LIN {X 0,Y 97.442,Z 457.914,A -85,B 0,C 180,E1 -28297.811,E2 -28297.811} C_VEL
LIN {X 0,Y 89.489,Z 462.022,A -85,B 0,C 180,E1 -28300.482,E2 -28300.482} C_VEL
LIN {X 0,Y 81.671,Z 465.606,A -85,B 0,C 180,E1 -28303.794,E2 -28303.794} C_VEL
LIN {X 0,Y 77.924,Z 467.495,A -85,B 0,C 180,E1 -28306.759,E2 -28306.759} C_VEL
LIN {X 0,Y 72.015,Z 470.678,A -85,B 0,C 180,E1 -28314.162,E2 -28314.162} C_VEL
LIN {X 0,Y 66.399,Z 473.568,A -85,B 0,C 180,E1 -28324.955,E2 -28324.955} C_VEL
LIN {X 0,Y 63.238,Z 475.299,A -85,B 0,C 180,E1 -28337.16,E2 -28337.16} C_VEL
LIN {X 0,Y 62.547,Z 475.896,A -85,B 0,C 180,E1 -28350.002,E2 -28350.002} C_VEL
LIN {X 0,Y 63.235,Z 475.326,A -85,B 0,C 180,E1 -28362.845,E2 -28362.845} C_VEL
LIN {X 0,Y 66.353,Z 473.633,A -85,B 0,C 180,E1 -28375.069,E2 -28375.069} C_VEL
LIN {X 0,Y 71.978,Z 470.774,A -85,B 0,C 180,E1 -28385.865,E2 -28385.865} C_VEL
LIN {X 0,Y 79.628,Z 466.628,A -85,B 0,C 180,E1 -28395.082,E2 -28395.082} C_VEL
LIN {X 0,Y 88.746,Z 461.261,A -85,B 0,C 180,E1 -28402.367,E2 -28402.367} C_VEL
LIN {X 0,Y 99.079,Z 454.353,A -85,B 0,C 180,E1 -28408.344,E2 -28408.344} C_VEL
LIN {X 0,Y 108.881,Z 446.931,A -85,B 0,C 180,E1 -28412.566,E2 -28412.566} C_VEL
LIN {X 0,Y 119.077,Z 437.984,A -85,B 0,C 180,E1 -28416.181,E2 -28416.181} C_VEL
LIN {X 0,Y 123.43,Z 433.764,A -85,B 0,C 180,E1 -28417.473,E2 -28417.473} C_VEL
LIN {X 0,Y 124.559,Z 432.45,A -85,B 0,C 180,E1 -28418.106,E2 -28418.106} C_VEL
LIN {X 0,Y 125.877,Z 428.922,A -85,B 0,C 180,E1 -28421.651,E2 -28421.651} C_VEL
LIN {X 0,Y 126.554,Z 427.011,A -85,B 0,C 180,E1 -28423.879,E2 -28423.879} C_VEL
LIN {X 0,Y 126.966,Z 424.818,A -85,B 0,C 180,E1 -28427.208,E2 -28427.208} C_VEL
LIN {X 0,Y 127.18,Z 423.255,A -85,B 0,C 180,E1 -28430.457,E2 -28430.457} C_VEL
LIN {X 0,Y 127.338,Z 422.165,A -85,B 0,C 180,E1 -28433.662,E2 -28433.662} C_VEL
LIN {X 0,Y 127.868,Z 420.898,A -85,B 0,C 180,E1 -28440,E2 -28440} C_VEL
LIN {X 0,Y 127.415,Z 422.493,A -85,B 0,C 180,E1 -28446.852,E2 -28446.852} C_VEL
LIN {X 0,Y 127.255,Z 423.571,A -85,B 0,C 180,E1 -28449.537,E2 -28449.537} C_VEL
LIN {X 0,Y 126.822,Z 425.492,A -85,B 0,C 180,E1 -28452.806,E2 -28452.806} C_VEL
LIN {X 0,Y 126.028,Z 428.183,A -85,B 0,C 180,E1 -28456.19,E2 -28456.19} C_VEL
LIN {X 0,Y 124.785,Z 431.569,A -85,B 0,C 180,E1 -28459.75,E2 -28459.75} C_VEL
LIN {X 0,Y 123.924,Z 433.592,A -85,B 0,C 180,E1 -28461.568,E2 -28461.568} C_VEL
LIN {X 0,Y 122.983,Z 434.784,A -85,B 0,C 180,E1 -28462.222,E2 -28462.222} C_VEL
LIN {X 0,Y 112.81,Z 444.196,A -85,B 0,C 180,E1 -28465.398,E2 -28465.398} C_VEL
LIN {X 0,Y 104.198,Z 451.23,A -85,B 0,C 180,E1 -28468.736,E2 -28468.736} C_VEL
LIN {X 0,Y 96.042,Z 457.197,A -85,B 0,C 180,E1 -28472.697,E2 -28472.697} C_VEL
LIN {X 0,Y 85.88,Z 463.77,A -85,B 0,C 180,E1 -28478.972,E2 -28478.972} C_VEL
LIN {X 0,Y 76.763,Z 469.049,A -85,B 0,C 180,E1 -28487.09,E2 -28487.09} C_VEL
LIN {X 0,Y 71.544,Z 471.892,A -85,B 0,C 180,E1 -28493.884,E2 -28493.884} C_VEL
LIN {X 0,Y 66.002,Z 474.79,A -85,B 0,C 180,E1 -28504.789,E2 -28504.789} C_VEL
LIN {X 0,Y 63.046,Z 476.52,A -85,B 0,C 180,E1 -28517.115,E2 -28517.115} C_VEL
LIN {X 0,Y 62.488,Z 477.112,A -85,B 0,C 180,E1 -28529.998,E2 -28529.998} C_VEL
LIN {X 0,Y 63.044,Z 476.499,A -85,B 0,C 180,E1 -28542.88,E2 -28542.88} C_VEL
LIN {X 0,Y 66.001,Z 474.741,A -85,B 0,C 180,E1 -28555.207,E2 -28555.207} C_VEL
LIN {X 0,Y 71.552,Z 471.819,A -85,B 0,C 180,E1 -28566.106,E2 -28566.106} C_VEL
LIN {X 0,Y 79.126,Z 467.663,A -85,B 0,C 180,E1 -28575.277,E2 -28575.277} C_VEL
LIN {X 0,Y 88.295,Z 462.161,A -85,B 0,C 180,E1 -28582.743,E2 -28582.743} C_VEL
LIN {X 0,Y 98.752,Z 455.167,A -85,B 0,C 180,E1 -28588.647,E2 -28588.647} C_VEL
LIN {X 0,Y 108.712,Z 447.473,A -85,B 0,C 180,E1 -28593.094,E2 -28593.094} C_VEL
LIN {X 0,Y 118.744,Z 438.664,A -85,B 0,C 180,E1 -28596.541,E2 -28596.541} C_VEL
LIN {X 0,Y 122.944,Z 434.565,A -85,B 0,C 180,E1 -28597.783,E2 -28597.783} C_VEL
LIN {X 0,Y 123.888,Z 433.395,A -85,B 0,C 180,E1 -28598.402,E2 -28598.402} C_VEL
LIN {X 0,Y 125.435,Z 429.38,A -85,B 0,C 180,E1 -28602.262,E2 -28602.262} C_VEL
LIN {X 0,Y 126.427,Z 426.495,A -85,B 0,C 180,E1 -28605.514,E2 -28605.514} C_VEL
LIN {X 0,Y 126.719,Z 425.289,A -85,B 0,C 180,E1 -28607.183,E2 -28607.183} C_VEL
LIN {X 0,Y 127.153,Z 423.361,A -85,B 0,C 180,E1 -28610.456,E2 -28610.456} C_VEL
LIN {X 0,Y 127.373,Z 422.07,A -85,B 0,C 180,E1 -28613.665,E2 -28613.665} C_VEL
LIN {X 0,Y 127.794,Z 420.619,A -85,B 0,C 180,E1 -28620,E2 -28620} C_VEL
LIN {X 0,Y 127.238,Z 421.924,A -85,B 0,C 180,E1 -28626.343,E2 -28626.343} C_VEL
LIN {X 0,Y 127.08,Z 423.01,A -85,B 0,C 180,E1 -28629.551,E2 -28629.551} C_VEL
LIN {X 0,Y 126.764,Z 425.502,A -85,B 0,C 180,E1 -28634.448,E2 -28634.448} C_VEL
LIN {X 0,Y 125.828,Z 428.596,A -85,B 0,C 180,E1 -28638.29,E2 -28638.29} C_VEL
LIN {X 0,Y 124.488,Z 432.184,A -85,B 0,C 180,E1 -28641.887,E2 -28641.887} C_VEL
LIN {X 0,Y 123.467,Z 433.483,A -85,B 0,C 180,E1 -28642.608,E2 -28642.608} C_VEL
LIN {X 0,Y 114.3,Z 442.123,A -85,B 0,C 180,E1 -28645.494,E2 -28645.494} C_VEL
LIN {X 0,Y 103.312,Z 451.121,A -85,B 0,C 180,E1 -28649.853,E2 -28649.853} C_VEL
LIN {X 0,Y 93.855,Z 457.813,A -85,B 0,C 180,E1 -28654.548,E2 -28654.548} C_VEL
LIN {X 0,Y 84.04,Z 464.002,A -85,B 0,C 180,E1 -28661.184,E2 -28661.184} C_VEL
LIN {X 0,Y 77.924,Z 467.495,A -85,B 0,C 180,E1 -28666.759,E2 -28666.759} C_VEL
LIN {X 0,Y 74.365,Z 469.237,A -85,B 0,C 180,E1 -28670.048,E2 -28670.048} C_VEL
LIN {X 0,Y 67.326,Z 471.662,A -85,B 0,C 180,E1 -28675.354,E2 -28675.354} C_VEL
LIN {X 0,Y 60.799,Z 473.558,A -85,B 0,C 180,E1 -28681.878,E2 -28681.878} C_VEL
LIN {X 0,Y 58.285,Z 474.398,A -85,B 0,C 180,E1 -28686.971,E2 -28686.971} C_VEL
LIN {X 0,Y 56.319,Z 475.368,A -85,B 0,C 180,E1 -28695.55,E2 -28695.55} C_VEL
LIN {X 0,Y 55.465,Z 475.965,A -85,B 0,C 180,E1 -28710.003,E2 -28710.003} C_VEL
LIN {X 0,Y 56.315,Z 475.395,A -85,B 0,C 180,E1 -28724.456,E2 -28724.456} C_VEL
LIN {X 0,Y 59.949,Z 473.702,A -85,B 0,C 180,E1 -28737.967,E2 -28737.967} C_VEL
LIN {X 0,Y 66.327,Z 470.843,A -85,B 0,C 180,E1 -28749.479,E2 -28749.479} C_VEL
LIN {X 0,Y 74.653,Z 466.753,A -85,B 0,C 180,E1 -28758.865,E2 -28758.865} C_VEL
LIN {X 0,Y 84.571,Z 461.329,A -85,B 0,C 180,E1 -28766.205,E2 -28766.205} C_VEL
LIN {X 0,Y 95.532,Z 454.42,A -85,B 0,C 180,E1 -28771.984,E2 -28771.984} C_VEL
LIN {X 0,Y 105.763,Z 446.999,A -85,B 0,C 180,E1 -28776.022,E2 -28776.022} C_VEL
LIN {X 0,Y 116.379,Z 438.051,A -85,B 0,C 180,E1 -28779.396,E2 -28779.396} C_VEL
LIN {X 0,Y 119.463,Z 435.151,A -85,B 0,C 180,E1 -28780.269,E2 -28780.269} C_VEL
LIN {X 0,Y 120.636,Z 432.702,A -85,B 0,C 180,E1 -28783.064,E2 -28783.064} C_VEL
LIN {X 0,Y 121.277,Z 431.216,A -85,B 0,C 180,E1 -28784.884,E2 -28784.884} C_VEL
LIN {X 0,Y 121.641,Z 430.076,A -85,B 0,C 180,E1 -28786.637,E2 -28786.637} C_VEL
LIN {X 0,Y 121.963,Z 428.494,A -85,B 0,C 180,E1 -28790.045,E2 -28790.045} C_VEL
LIN {X 0,Y 122.275,Z 427.316,A -85,B 0,C 180,E1 -28793.399,E2 -28793.399} C_VEL
LIN {X 0,Y 122.896,Z 426.011,A -85,B 0,C 180,E1 -28800,E2 -28800} C_VEL
LIN {X 0,Y 122.378,Z 427.479,A -85,B 0,C 180,E1 -28806.595,E2 -28806.595} C_VEL
LIN {X 0,Y 121.745,Z 429.512,A -85,B 0,C 180,E1 -28811.077,E2 -28811.077} C_VEL
LIN {X 0,Y 121.308,Z 430.918,A -85,B 0,C 180,E1 -28813.399,E2 -28813.399} C_VEL
LIN {X 0,Y 119.986,Z 433.936,A -85,B 0,C 180,E1 -28817.029,E2 -28817.029} C_VEL
LIN {X 0,Y 119.037,Z 435.896,A -85,B 0,C 180,E1 -28819.152,E2 -28819.152} C_VEL
LIN {X 0,Y 117.658,Z 437.389,A -85,B 0,C 180,E1 -28819.815,E2 -28819.815} C_VEL
LIN {X 0,Y 106.892,Z 446.596,A -85,B 0,C 180,E1 -28823.003,E2 -28823.003} C_VEL
LIN {X 0,Y 96.663,Z 454.257,A -85,B 0,C 180,E1 -28827.043,E2 -28827.043} C_VEL
LIN {X 0,Y 86.828,Z 460.604,A -85,B 0,C 180,E1 -28831.799,E2 -28831.799} C_VEL
LIN {X 0,Y 76.579,Z 466.441,A -85,B 0,C 180,E1 -28838.73,E2 -28838.73} C_VEL
LIN {X 0,Y 69.824,Z 469.915,A -85,B 0,C 180,E1 -28845.203,E2 -28845.203} C_VEL
LIN {X 0,Y 62.467,Z 473.422,A -85,B 0,C 180,E1 -28855.766,E2 -28855.766} C_VEL
LIN {X 0,Y 57.49,Z 475.729,A -85,B 0,C 180,E1 -28868.483,E2 -28868.483} C_VEL
LIN {X 0,Y 55.392,Z 476.889,A -85,B 0,C 180,E1 -28882.708,E2 -28882.708} C_VEL
LIN {X 0,Y 55.387,Z 477.043,A -85,B 0,C 180,E1 -28889.997,E2 -28889.997} C_VEL
LIN {X 0,Y 56.105,Z 476.429,A -85,B 0,C 180,E1 -28904.506,E2 -28904.506} C_VEL
LIN {X 0,Y 59.603,Z 474.671,A -85,B 0,C 180,E1 -28918.138,E2 -28918.138} C_VEL
LIN {X 0,Y 65.896,Z 471.749,A -85,B 0,C 180,E1 -28929.781,E2 -28929.781} C_VEL
LIN {X 0,Y 74.266,Z 467.592,A -85,B 0,C 180,E1 -28939.202,E2 -28939.202} C_VEL
LIN {X 0,Y 84.154,Z 462.09,A -85,B 0,C 180,E1 -28946.625,E2 -28946.625} C_VEL
LIN {X 0,Y 95.235,Z 455.096,A -85,B 0,C 180,E1 -28952.315,E2 -28952.315} C_VEL
LIN {X 0,Y 104.959,Z 447.945,A -85,B 0,C 180,E1 -28956.312,E2 -28956.312} C_VEL
LIN {X 0,Y 116.087,Z 438.592,A -85,B 0,C 180,E1 -28959.776,E2 -28959.776} C_VEL
LIN {X 0,Y 117.64,Z 437.143,A -85,B 0,C 180,E1 -28960.201,E2 -28960.201} C_VEL
LIN {X 0,Y 118.973,Z 435.649,A -85,B 0,C 180,E1 -28960.93,E2 -28960.93} C_VEL
LIN {X 0,Y 120.601,Z 432.176,A -85,B 0,C 180,E1 -28964.798,E2 -28964.798} C_VEL
LIN {X 0,Y 121.203,Z 430.735,A -85,B 0,C 180,E1 -28966.589,E2 -28966.589} C_VEL
LIN {X 0,Y 121.854,Z 428.703,A -85,B 0,C 180,E1 -28970.036,E2 -28970.036} C_VEL
LIN {X 0,Y 122.294,Z 427.252,A -85,B 0,C 180,E1 -28973.4,E2 -28973.4} C_VEL
LIN {X 0,Y 122.823,Z 425.753,A -85,B 0,C 180,E1 -28980,E2 -28980} C_VEL
LIN {X 0,Y 122.169,Z 427.091,A -85,B 0,C 180,E1 -28986.607,E2 -28986.607} C_VEL
LIN {X 0,Y 121.743,Z 428.758,A -85,B 0,C 180,E1 -28991.085,E2 -28991.085} C_VEL
LIN {X 0,Y 121.552,Z 429.836,A -85,B 0,C 180,E1 -28993.373,E2 -28993.373} C_VEL
LIN {X 0,Y 120.585,Z 432.443,A -85,B 0,C 180,E1 -28996.943,E2 -28996.943} C_VEL
LIN {X 0,Y 119.411,Z 434.854,A -85,B 0,C 180,E1 -28999.67,E2 -28999.67} C_VEL
LIN {X 0,Y 116.428,Z 437.778,A -85,B 0,C 180,E1 -29000.675,E2 -29000.675} C_VEL
LIN {X 0,Y 105.837,Z 446.761,A -85,B 0,C 180,E1 -29004.075,E2 -29004.075} C_VEL
LIN {X 0,Y 95.571,Z 454.208,A -85,B 0,C 180,E1 -29008.066,E2 -29008.066} C_VEL
LIN {X 0,Y 84.625,Z 461.165,A -85,B 0,C 180,E1 -29013.856,E2 -29013.856} C_VEL
LIN {X 0,Y 74.274,Z 466.832,A -85,B 0,C 180,E1 -29021.481,E2 -29021.481} C_VEL
LIN {X 0,Y 66.361,Z 470.748,A -85,B 0,C 180,E1 -29030.552,E2 -29030.552} C_VEL
LIN {X 0,Y 59.992,Z 473.638,A -85,B 0,C 180,E1 -29042.06,E2 -29042.06} C_VEL
LIN {X 0,Y 58.285,Z 474.398,A -85,B 0,C 180,E1 -29046.971,E2 -29046.971} C_VEL
LIN {X 0,Y 56.244,Z 475.136,A -85,B 0,C 180,E1 -29052.47,E2 -29052.47} C_VEL
LIN {X 0,Y 53.738,Z 475.668,A -85,B 0,C 180,E1 -29058.065,E2 -29058.065} C_VEL
LIN {X 0,Y 49.32,Z 476.068,A -85,B 0,C 180,E1 -29070.536,E2 -29070.536} C_VEL
LIN {X 0,Y 48.601,Z 475.81,A -85,B 0,C 180,E1 -29079.882,E2 -29079.882} C_VEL
LIN {X 0,Y 51.219,Z 474.76,A -85,B 0,C 180,E1 -29094.311,E2 -29094.311} C_VEL
LIN {X 0,Y 57.045,Z 472.491,A -85,B 0,C 180,E1 -29108.027,E2 -29108.027} C_VEL
LIN {X 0,Y 65.36,Z 469.026,A -85,B 0,C 180,E1 -29118.827,E2 -29118.827} C_VEL
LIN {X 0,Y 75.354,Z 464.284,A -85,B 0,C 180,E1 -29127.079,E2 -29127.079} C_VEL
LIN {X 0,Y 86.504,Z 458.141,A -85,B 0,C 180,E1 -29133.343,E2 -29133.343} C_VEL
LIN {X 0,Y 98.494,Z 450.406,A -85,B 0,C 180,E1 -29138.068,E2 -29138.068} C_VEL
LIN {X 0,Y 109.411,Z 442.08,A -85,B 0,C 180,E1 -29141.538,E2 -29141.538} C_VEL
LIN {X 0,Y 114.064,Z 438.118,A -85,B 0,C 180,E1 -29142.752,E2 -29142.752} C_VEL
LIN {X 0,Y 115.111,Z 436.741,A -85,B 0,C 180,E1 -29144.021,E2 -29144.021} C_VEL
LIN {X 0,Y 115.899,Z 435.266,A -85,B 0,C 180,E1 -29145.985,E2 -29145.985} C_VEL
LIN {X 0,Y 116.535,Z 433.504,A -85,B 0,C 180,E1 -29149.576,E2 -29149.576} C_VEL
LIN {X 0,Y 116.94,Z 432.294,A -85,B 0,C 180,E1 -29153.096,E2 -29153.096} C_VEL
LIN {X 0,Y 117.708,Z 430.931,A -85,B 0,C 180,E1 -29160,E2 -29160} C_VEL
LIN {X 0,Y 117.302,Z 431.567,A -85,B 0,C 180,E1 -29163.434,E2 -29163.434} C_VEL
LIN {X 0,Y 117.008,Z 432.494,A -85,B 0,C 180,E1 -29166.899,E2 -29166.899} C_VEL
LIN {X 0,Y 116.402,Z 434.014,A -85,B 0,C 180,E1 -29170.435,E2 -29170.435} C_VEL
LIN {X 0,Y 115.253,Z 436.366,A -85,B 0,C 180,E1 -29174.117,E2 -29174.117} C_VEL
LIN {X 0,Y 113.826,Z 438.748,A -85,B 0,C 180,E1 -29176.857,E2 -29176.857} C_VEL
LIN {X 0,Y 102.087,Z 448.202,A -85,B 0,C 180,E1 -29180.041,E2 -29180.041} C_VEL
LIN {X 0,Y 92.127,Z 455.199,A -85,B 0,C 180,E1 -29183.731,E2 -29183.731} C_VEL
LIN {X 0,Y 80.455,Z 462.152,A -85,B 0,C 180,E1 -29189.127,E2 -29189.127} C_VEL
LIN {X 0,Y 69.762,Z 467.619,A -85,B 0,C 180,E1 -29196.296,E2 -29196.296} C_VEL
LIN {X 0,Y 60.555,Z 471.754,A -85,B 0,C 180,E1 -29205.861,E2 -29205.861} C_VEL
LIN {X 0,Y 53.399,Z 474.652,A -85,B 0,C 180,E1 -29218.231,E2 -29218.231} C_VEL
LIN {X 0,Y 49.236,Z 476.382,A -85,B 0,C 180,E1 -29233.409,E2 -29233.409} C_VEL
LIN {X 0,Y 48.302,Z 476.974,A -85,B 0,C 180,E1 -29249.997,E2 -29249.997} C_VEL
LIN {X 0,Y 49.234,Z 476.36,A -85,B 0,C 180,E1 -29266.585,E2 -29266.585} C_VEL
LIN {X 0,Y 53.398,Z 474.601,A -85,B 0,C 180,E1 -29281.762,E2 -29281.762} C_VEL
LIN {X 0,Y 60.563,Z 471.678,A -85,B 0,C 180,E1 -29294.123,E2 -29294.123} C_VEL
LIN {X 0,Y 69.785,Z 467.521,A -85,B 0,C 180,E1 -29303.671,E2 -29303.671} C_VEL
LIN {X 0,Y 80.444,Z 462.019,A -85,B 0,C 180,E1 -29310.881,E2 -29310.881} C_VEL
LIN {X 0,Y 92.136,Z 455.025,A -85,B 0,C 180,E1 -29316.249,E2 -29316.249} C_VEL
LIN {X 0,Y 102.321,Z 447.858,A -85,B 0,C 180,E1 -29319.985,E2 -29319.985} C_VEL
LIN {X 0,Y 113.81,Z 438.52,A -85,B 0,C 180,E1 -29323.16,E2 -29323.16} C_VEL
LIN {X 0,Y 115.17,Z 436.18,A -85,B 0,C 180,E1 -29325.872,E2 -29325.872} C_VEL
LIN {X 0,Y 116.316,Z 433.825,A -85,B 0,C 180,E1 -29329.557,E2 -29329.557} C_VEL
LIN {X 0,Y 116.922,Z 432.282,A -85,B 0,C 180,E1 -29333.096,E2 -29333.096} C_VEL
LIN {X 0,Y 117.224,Z 431.342,A -85,B 0,C 180,E1 -29336.563,E2 -29336.563} C_VEL
LIN {X 0,Y 117.643,Z 430.687,A -85,B 0,C 180,E1 -29340,E2 -29340} C_VEL
LIN {X 0,Y 117.199,Z 431.223,A -85,B 0,C 180,E1 -29343.438,E2 -29343.438} C_VEL
LIN {X 0,Y 116.774,Z 432.227,A -85,B 0,C 180,E1 -29347.384,E2 -29347.384} C_VEL
LIN {X 0,Y 116.446,Z 433.29,A -85,B 0,C 180,E1 -29350.432,E2 -29350.432} C_VEL
LIN {X 0,Y 115.774,Z 435.089,A -85,B 0,C 180,E1 -29354.053,E2 -29354.053} C_VEL
LIN {X 0,Y 115.098,Z 436.427,A -85,B 0,C 180,E1 -29355.918,E2 -29355.918} C_VEL
LIN {X 0,Y 114.105,Z 437.849,A -85,B 0,C 180,E1 -29357.322,E2 -29357.322} C_VEL
LIN {X 0,Y 103.117,Z 446.833,A -85,B 0,C 180,E1 -29360.43,E2 -29360.43} C_VEL
LIN {X 0,Y 92.433,Z 454.279,A -85,B 0,C 180,E1 -29364.167,E2 -29364.167} C_VEL
LIN {X 0,Y 80.862,Z 461.235,A -85,B 0,C 180,E1 -29369.647,E2 -29369.647} C_VEL
LIN {X 0,Y 69.109,Z 467.216,A -85,B 0,C 180,E1 -29377.603,E2 -29377.603} C_VEL
LIN {X 0,Y 61.009,Z 470.818,A -85,B 0,C 180,E1 -29386.281,E2 -29386.281} C_VEL
LIN {X 0,Y 53.778,Z 473.708,A -85,B 0,C 180,E1 -29398.487,E2 -29398.487} C_VEL
LIN {X 0,Y 49.467,Z 475.437,A -85,B 0,C 180,E1 -29413.496,E2 -29413.496} C_VEL
LIN {X 0,Y 48.366,Z 476.034,A -85,B 0,C 180,E1 -29430.003,E2 -29430.003} C_VEL
LIN {X 0,Y 48.601,Z 475.81,A -85,B 0,C 180,E1 -29439.882,E2 -29439.882} C_VEL
LIN {X 0,Y 48.791,Z 475.476,A -85,B 0,C 180,E1 -29446.811,E2 -29446.811} C_VEL
LIN {X 0,Y 48.736,Z 474.556,A -85,B 0,C 180,E1 -29458.432,E2 -29458.432} C_VEL
LIN {X 0,Y 49.871,Z 473.469,A -85,B 0,C 180,E1 -29467.532,E2 -29467.532} C_VEL
LIN {X 0,Y 52.152,Z 472.394,A -85,B 0,C 180,E1 -29473.57,E2 -29473.57} C_VEL
LIN {X 0,Y 53.248,Z 471.951,A -85,B 0,C 180,E1 -29475.304,E2 -29475.304} C_VEL
LIN {X 0,Y 64.288,Z 467.695,A -85,B 0,C 180,E1 -29486.865,E2 -29486.865} C_VEL
LIN {X 0,Y 74.601,Z 462.935,A -85,B 0,C 180,E1 -29493.508,E2 -29493.508} C_VEL
LIN {X 0,Y 86.607,Z 456.407,A -85,B 0,C 180,E1 -29498.943,E2 -29498.943} C_VEL
LIN {X 0,Y 97.634,Z 449.361,A -85,B 0,C 180,E1 -29502.513,E2 -29502.513} C_VEL
LIN {X 0,Y 108.881,Z 440.887,A -85,B 0,C 180,E1 -29505.518,E2 -29505.518} C_VEL
LIN {X 0,Y 110.441,Z 439.109,A -85,B 0,C 180,E1 -29507.366,E2 -29507.366} C_VEL
LIN {X 0,Y 111.392,Z 437.043,A -85,B 0,C 180,E1 -29512.75,E2 -29512.75} C_VEL
LIN {X 0,Y 111.809,Z 436.191,A -85,B 0,C 180,E1 -29516.396,E2 -29516.396} C_VEL
LIN {X 0,Y 112.331,Z 435.629,A -85,B 0,C 180,E1 -29520,E2 -29520} C_VEL
LIN {X 0,Y 111.864,Z 436.276,A -85,B 0,C 180,E1 -29523.602,E2 -29523.602} C_VEL
LIN {X 0,Y 111.369,Z 437.326,A -85,B 0,C 180,E1 -29527.25,E2 -29527.25} C_VEL
LIN {X 0,Y 110.443,Z 439.039,A -85,B 0,C 180,E1 -29531.005,E2 -29531.005} C_VEL
LIN {X 0,Y 109.775,Z 440.135,A -85,B 0,C 180,E1 -29532.843,E2 -29532.843} C_VEL
LIN {X 0,Y 108.673,Z 441.392,A -85,B 0,C 180,E1 -29534.052,E2 -29534.052} C_VEL
LIN {X 0,Y 98.011,Z 449.416,A -85,B 0,C 180,E1 -29536.668,E2 -29536.668} C_VEL
LIN {X 0,Y 86.374,Z 456.993,A -85,B 0,C 180,E1 -29540.652,E2 -29540.652} C_VEL
LIN {X 0,Y 74.273,Z 463.564,A -85,B 0,C 180,E1 -29545.979,E2 -29545.979} C_VEL
LIN {X 0,Y 63.083,Z 468.707,A -85,B 0,C 180,E1 -29553.328,E2 -29553.328} C_VEL
LIN {X 0,Y 55.637,Z 471.685,A -85,B 0,C 180,E1 -29560.716,E2 -29560.716} C_VEL
LIN {X 0,Y 47.467,Z 474.583,A -85,B 0,C 180,E1 -29573.681,E2 -29573.681} C_VEL
LIN {X 0,Y 42.433,Z 476.312,A -85,B 0,C 180,E1 -29590.652,E2 -29590.652} C_VEL
LIN {X 0,Y 41.187,Z 476.905,A -85,B 0,C 180,E1 -29609.996,E2 -29609.996} C_VEL
LIN {X 0,Y 42.431,Z 476.29,A -85,B 0,C 180,E1 -29629.341,E2 -29629.341} C_VEL
LIN {X 0,Y 47.466,Z 474.531,A -85,B 0,C 180,E1 -29646.312,E2 -29646.312} C_VEL
LIN {X 0,Y 55.644,Z 471.608,A -85,B 0,C 180,E1 -29659.267,E2 -29659.267} C_VEL
LIN {X 0,Y 65.794,Z 467.451,A -85,B 0,C 180,E1 -29668.703,E2 -29668.703} C_VEL
LIN {X 0,Y 77.213,Z 461.948,A -85,B 0,C 180,E1 -29675.527,E2 -29675.527} C_VEL
LIN {X 0,Y 89.496,Z 454.953,A -85,B 0,C 180,E1 -29680.441,E2 -29680.441} C_VEL
LIN {X 0,Y 99.751,Z 448.032,A -85,B 0,C 180,E1 -29683.729,E2 -29683.729} C_VEL
LIN {X 0,Y 108.665,Z 441.16,A -85,B 0,C 180,E1 -29685.953,E2 -29685.953} C_VEL
LIN {X 0,Y 109.77,Z 439.864,A -85,B 0,C 180,E1 -29687.267,E2 -29687.267} C_VEL
LIN {X 0,Y 110.371,Z 438.856,A -85,B 0,C 180,E1 -29688.988,E2 -29688.988} C_VEL
LIN {X 0,Y 111.297,Z 437.121,A -85,B 0,C 180,E1 -29692.745,E2 -29692.745} C_VEL
LIN {X 0,Y 111.779,Z 436.077,A -85,B 0,C 180,E1 -29696.396,E2 -29696.396} C_VEL
LIN {X 0,Y 112.264,Z 435.409,A -85,B 0,C 180,E1 -29700,E2 -29700} C_VEL
LIN {X 0,Y 111.758,Z 435.954,A -85,B 0,C 180,E1 -29703.606,E2 -29703.606} C_VEL
LIN {X 0,Y 111.31,Z 436.827,A -85,B 0,C 180,E1 -29707.255,E2 -29707.255} C_VEL
LIN {X 0,Y 110.697,Z 438.178,A -85,B 0,C 180,E1 -29710.98,E2 -29710.98} C_VEL
LIN {X 0,Y 110.1,Z 439.348,A -85,B 0,C 180,E1 -29713.423,E2 -29713.423} C_VEL
LIN {X 0,Y 108.919,Z 440.621,A -85,B 0,C 180,E1 -29714.571,E2 -29714.571} C_VEL
LIN {X 0,Y 97.678,Z 449.135,A -85,B 0,C 180,E1 -29717.579,E2 -29717.579} C_VEL
LIN {X 0,Y 86.636,Z 456.222,A -85,B 0,C 180,E1 -29721.117,E2 -29721.117} C_VEL
LIN {X 0,Y 74.642,Z 462.795,A -85,B 0,C 180,E1 -29726.565,E2 -29726.565} C_VEL
LIN {X 0,Y 64.305,Z 467.584,A -85,B 0,C 180,E1 -29733.125,E2 -29733.125} C_VEL
LIN {X 0,Y 56.051,Z 470.889,A -85,B 0,C 180,E1 -29741.214,E2 -29741.214} C_VEL
LIN {X 0,Y 47.828,Z 473.778,A -85,B 0,C 180,E1 -29754.006,E2 -29754.006} C_VEL
LIN {X 0,Y 42.676,Z 475.507,A -85,B 0,C 180,E1 -29770.774,E2 -29770.774} C_VEL
LIN {X 0,Y 41.282,Z 476.103,A -85,B 0,C 180,E1 -29790.004,E2 -29790.004} C_VEL
LIN {X 0,Y 42.67,Z 475.533,A -85,B 0,C 180,E1 -29809.237,E2 -29809.237} C_VEL
LIN {X 0,Y 47.792,Z 473.84,A -85,B 0,C 180,E1 -29826.034,E2 -29826.034} C_VEL
LIN {X 0,Y 53.248,Z 471.951,A -85,B 0,C 180,E1 -29835.304,E2 -29835.304} C_VEL
LIN {X 0,Y 56.427,Z 470.681,A -85,B 0,C 180,E1 -29840.325,E2 -29840.325} C_VEL
LIN {X 0,Y 61.102,Z 468.246,A -85,B 0,C 180,E1 -29848.542,E2 -29848.542} C_VEL
LIN {X 0,Y 65.43,Z 465.999,A -85,B 0,C 180,E1 -29854.243,E2 -29854.243} C_VEL
LIN {X 0,Y 69.487,Z 464.048,A -85,B 0,C 180,E1 -29857.503,E2 -29857.503} C_VEL
LIN {X 0,Y 71.024,Z 463.312,A -85,B 0,C 180,E1 -29858.326,E2 -29858.326} C_VEL
LIN {X 0,Y 84.311,Z 456.474,A -85,B 0,C 180,E1 -29863.462,E2 -29863.462} C_VEL
LIN {X 0,Y 95.659,Z 449.473,A -85,B 0,C 180,E1 -29866.596,E2 -29866.596} C_VEL
LIN {X 0,Y 103.972,Z 443.547,A -85,B 0,C 180,E1 -29868.553,E2 -29868.553} C_VEL
LIN {X 0,Y 105.224,Z 442.266,A -85,B 0,C 180,E1 -29870.387,E2 -29870.387} C_VEL
LIN {X 0,Y 106.156,Z 440.691,A -85,B 0,C 180,E1 -29876.204,E2 -29876.204} C_VEL
LIN {X 0,Y 106.764,Z 440.109,A -85,B 0,C 180,E1 -29880,E2 -29880} C_VEL
LIN {X 0,Y 105.904,Z 441.239,A -85,B 0,C 180,E1 -29885.476,E2 -29885.476} C_VEL
LIN {X 0,Y 104.967,Z 442.74,A -85,B 0,C 180,E1 -29889.423,E2 -29889.423} C_VEL
LIN {X 0,Y 103.812,Z 443.926,A -85,B 0,C 180,E1 -29890.995,E2 -29890.995} C_VEL
LIN {X 0,Y 92.21,Z 452.031,A -85,B 0,C 180,E1 -29893.644,E2 -29893.644} C_VEL
LIN {X 0,Y 80.888,Z 458.737,A -85,B 0,C 180,E1 -29897.106,E2 -29897.106} C_VEL
LIN {X 0,Y 68.348,Z 464.923,A -85,B 0,C 180,E1 -29902.261,E2 -29902.261} C_VEL
LIN {X 0,Y 56.139,Z 469.892,A -85,B 0,C 180,E1 -29910.049,E2 -29910.049} C_VEL
LIN {X 0,Y 46.319,Z 473.215,A -85,B 0,C 180,E1 -29920.65,E2 -29920.65} C_VEL
LIN {X 0,Y 38.35,Z 475.521,A -85,B 0,C 180,E1 -29936.644,E2 -29936.644} C_VEL
LIN {X 0,Y 34.326,Z 476.682,A -85,B 0,C 180,E1 -29958.181,E2 -29958.181} C_VEL
LIN {X 0,Y 34.08,Z 476.836,A -85,B 0,C 180,E1 -29969.995,E2 -29969.995} C_VEL
LIN {X 0,Y 35.775,Z 476.22,A -85,B 0,C 180,E1 -29993.13,E2 -29993.13} C_VEL
LIN {X 0,Y 41.923,Z 474.461,A -85,B 0,C 180,E1 -30012.105,E2 -30012.105} C_VEL
LIN {X 0,Y 51.261,Z 471.538,A -85,B 0,C 180,E1 -30025.34,E2 -30025.34} C_VEL
LIN {X 0,Y 62.37,Z 467.38,A -85,B 0,C 180,E1 -30034.343,E2 -30034.343} C_VEL
LIN {X 0,Y 74.527,Z 461.877,A -85,B 0,C 180,E1 -30040.555,E2 -30040.555} C_VEL
LIN {X 0,Y 87.36,Z 454.882,A -85,B 0,C 180,E1 -30044.869,E2 -30044.869} C_VEL
LIN {X 0,Y 99.049,Z 447.233,A -85,B 0,C 180,E1 -30047.98,E2 -30047.98} C_VEL
LIN {X 0,Y 103.744,Z 443.754,A -85,B 0,C 180,E1 -30049.001,E2 -30049.001} C_VEL
LIN {X 0,Y 104.899,Z 442.561,A -85,B 0,C 180,E1 -30050.55,E2 -30050.55} C_VEL
LIN {X 0,Y 105.873,Z 440.994,A -85,B 0,C 180,E1 -30054.67,E2 -30054.67} C_VEL
LIN {X 0,Y 106.695,Z 439.911,A -85,B 0,C 180,E1 -30060,E2 -30060} C_VEL
LIN {X 0,Y 105.882,Z 440.796,A -85,B 0,C 180,E1 -30065.38,E2 -30065.38} C_VEL
LIN {X 0,Y 104.938,Z 442.443,A -85,B 0,C 180,E1 -30070.613,E2 -30070.613} C_VEL
LIN {X 0,Y 102.528,Z 444.398,A -85,B 0,C 180,E1 -30071.868,E2 -30071.868} C_VEL
LIN {X 0,Y 90.845,Z 452.41,A -85,B 0,C 180,E1 -30074.762,E2 -30074.762} C_VEL
LIN {X 0,Y 77.963,Z 459.769,A -85,B 0,C 180,E1 -30078.832,E2 -30078.832} C_VEL
LIN {X 0,Y 65.646,Z 465.604,A -85,B 0,C 180,E1 -30084.502,E2 -30084.502} C_VEL
LIN {X 0,Y 56.977,Z 469.06,A -85,B 0,C 180,E1 -30090.303,E2 -30090.303} C_VEL
LIN {X 0,Y 46.655,Z 472.552,A -85,B 0,C 180,E1 -30101.139,E2 -30101.139} C_VEL
LIN {X 0,Y 38.675,Z 474.854,A -85,B 0,C 180,E1 -30116.97,E2 -30116.97} C_VEL
LIN {X 0,Y 34.493,Z 476.019,A -85,B 0,C 180,E1 -30138.248,E2 -30138.248} C_VEL
LIN {X 0,Y 34.171,Z 476.172,A -85,B 0,C 180,E1 -30150.005,E2 -30150.005} C_VEL
LIN {X 0,Y 36.019,Z 475.602,A -85,B 0,C 180,E1 -30172.973,E2 -30172.973} C_VEL
LIN {X 0,Y 42.223,Z 473.909,A -85,B 0,C 180,E1 -30191.748,E2 -30191.748} C_VEL
LIN {X 0,Y 51.589,Z 471.05,A -85,B 0,C 180,E1 -30204.828,E2 -30204.828} C_VEL
LIN {X 0,Y 62.666,Z 466.958,A -85,B 0,C 180,E1 -30213.797,E2 -30213.797} C_VEL
LIN {X 0,Y 71.024,Z 463.312,A -85,B 0,C 180,E1 -30218.326,E2 -30218.326} C_VEL
LIN {X 0,Y 75.479,Z 461.113,A -85,B 0,C 180,E1 -30220.817,E2 -30220.817} C_VEL
LIN {X 0,Y 82.175,Z 457.277,A -85,B 0,C 180,E1 -30225.335,E2 -30225.335} C_VEL
LIN {X 0,Y 89.027,Z 452.971,A -85,B 0,C 180,E1 -30229.177,E2 -30229.177} C_VEL
LIN {X 0,Y 93.553,Z 450.006,A -85,B 0,C 180,E1 -30230.681,E2 -30230.681} C_VEL
LIN {X 0,Y 99.392,Z 446.069,A -85,B 0,C 180,E1 -30231.87,E2 -30231.87} C_VEL
LIN {X 0,Y 100.324,Z 444.955,A -85,B 0,C 180,E1 -30235.983,E2 -30235.983} C_VEL
LIN {X 0,Y 100.992,Z 444.381,A -85,B 0,C 180,E1 -30240,E2 -30240} C_VEL
LIN {X 0,Y 100.333,Z 445.081,A -85,B 0,C 180,E1 -30244.016,E2 -30244.016} C_VEL
LIN {X 0,Y 99.271,Z 446.326,A -85,B 0,C 180,E1 -30247.624,E2 -30247.624} C_VEL
LIN {X 0,Y 87.425,Z 453.983,A -85,B 0,C 180,E1 -30250.01,E2 -30250.01} C_VEL
LIN {X 0,Y 75.762,Z 460.331,A -85,B 0,C 180,E1 -30253.084,E2 -30253.084} C_VEL
LIN {X 0,Y 62.772,Z 466.167,A -85,B 0,C 180,E1 -30257.882,E2 -30257.882} C_VEL
LIN {X 0,Y 52.123,Z 470.105,A -85,B 0,C 180,E1 -30263.859,E2 -30263.859} C_VEL
LIN {X 0,Y 41.999,Z 473.146,A -85,B 0,C 180,E1 -30273.203,E2 -30273.203} C_VEL
LIN {X 0,Y 32.607,Z 475.452,A -85,B 0,C 180,E1 -30289.708,E2 -30289.708} C_VEL
LIN {X 0,Y 27.388,Z 476.613,A -85,B 0,C 180,E1 -30315.125,E2 -30315.125} C_VEL
LIN {X 0,Y 26.986,Z 476.767,A -85,B 0,C 180,E1 -30329.994,E2 -30329.994} C_VEL
LIN {X 0,Y 29.352,Z 476.151,A -85,B 0,C 180,E1 -30358.606,E2 -30358.606} C_VEL
LIN {X 0,Y 36.938,Z 474.391,A -85,B 0,C 180,E1 -30379.551,E2 -30379.551} C_VEL
LIN {X 0,Y 47.556,Z 471.467,A -85,B 0,C 180,E1 -30392.453,E2 -30392.453} C_VEL
LIN {X 0,Y 59.616,Z 467.309,A -85,B 0,C 180,E1 -30400.569,E2 -30400.569} C_VEL
LIN {X 0,Y 72.457,Z 461.806,A -85,B 0,C 180,E1 -30405.908,E2 -30405.908} C_VEL
LIN {X 0,Y 85.765,Z 454.811,A -85,B 0,C 180,E1 -30409.512,E2 -30409.512} C_VEL
LIN {X 0,Y 97.622,Z 447.292,A -85,B 0,C 180,E1 -30412.053,E2 -30412.053} C_VEL
LIN {X 0,Y 99.273,Z 446.105,A -85,B 0,C 180,E1 -30412.341,E2 -30412.341} C_VEL
LIN {X 0,Y 100.273,Z 444.896,A -85,B 0,C 180,E1 -30415.981,E2 -30415.981} C_VEL
LIN {X 0,Y 100.942,Z 444.184,A -85,B 0,C 180,E1 -30420,E2 -30420} C_VEL
LIN {X 0,Y 100.293,Z 444.741,A -85,B 0,C 180,E1 -30424.019,E2 -30424.019} C_VEL
LIN {X 0,Y 99.415,Z 445.83,A -85,B 0,C 180,E1 -30428.242,E2 -30428.242} C_VEL
LIN {X 0,Y 87.615,Z 453.486,A -85,B 0,C 180,E1 -30430.708,E2 -30430.708} C_VEL
LIN {X 0,Y 75.955,Z 459.84,A -85,B 0,C 180,E1 -30433.712,E2 -30433.712} C_VEL
LIN {X 0,Y 63.02,Z 465.675,A -85,B 0,C 180,E1 -30438.582,E2 -30438.582} C_VEL
LIN {X 0,Y 53.716,Z 469.13,A -85,B 0,C 180,E1 -30443.683,E2 -30443.683} C_VEL
LIN {X 0,Y 42.296,Z 472.622,A -85,B 0,C 180,E1 -30453.825,E2 -30453.825} C_VEL
LIN {X 0,Y 32.925,Z 474.924,A -85,B 0,C 180,E1 -30470.189,E2 -30470.189} C_VEL
LIN {X 0,Y 27.562,Z 476.088,A -85,B 0,C 180,E1 -30495.233,E2 -30495.233} C_VEL
LIN {X 0,Y 27.066,Z 476.241,A -85,B 0,C 180,E1 -30510.006,E2 -30510.006} C_VEL
LIN {X 0,Y 29.598,Z 475.671,A -85,B 0,C 180,E1 -30538.358,E2 -30538.358} C_VEL
LIN {X 0,Y 37.197,Z 473.978,A -85,B 0,C 180,E1 -30559.098,E2 -30559.098} C_VEL
LIN {X 0,Y 47.822,Z 471.118,A -85,B 0,C 180,E1 -30571.862,E2 -30571.862} C_VEL
LIN {X 0,Y 59.852,Z 467.027,A -85,B 0,C 180,E1 -30579.953,E2 -30579.953} C_VEL
LIN {X 0,Y 72.661,Z 461.602,A -85,B 0,C 180,E1 -30585.297,E2 -30585.297} C_VEL
LIN {X 0,Y 82.562,Z 456.542,A -85,B 0,C 180,E1 -30588.219,E2 -30588.219} C_VEL
LIN {X 0,Y 93.553,Z 450.006,A -85,B 0,C 180,E1 -30590.681,E2 -30590.681} C_VEL
LIN {X 0,Y 94.657,Z 449.191,A -85,B 0,C 180,E1 -30591.504,E2 -30591.504} C_VEL
LIN {X 0,Y 95.041,Z 448.74,A -85,B 0,C 180,E1 -30593.181,E2 -30593.181} C_VEL
LIN {X 0,Y 94.556,Z 448.737,A -85,B 0,C 180,E1 -30597.853,E2 -30597.853} C_VEL
LIN {X 0,Y 95.04,Z 448.42,A -85,B 0,C 180,E1 -30600,E2 -30600} C_VEL
LIN {X 0,Y 94.5,Z 448.907,A -85,B 0,C 180,E1 -30603.197,E2 -30603.197} C_VEL
LIN {X 0,Y 91.638,Z 450.822,A -85,B 0,C 180,E1 -30604.423,E2 -30604.423} C_VEL
LIN {X 0,Y 77.893,Z 458.601,A -85,B 0,C 180,E1 -30607.021,E2 -30607.021} C_VEL
LIN {X 0,Y 64.307,Z 464.786,A -85,B 0,C 180,E1 -30610.383,E2 -30610.383} C_VEL
LIN {X 0,Y 48.841,Z 470.296,A -85,B 0,C 180,E1 -30616.725,E2 -30616.725} C_VEL
LIN {X 0,Y 38.541,Z 473.077,A -85,B 0,C 180,E1 -30624.244,E2 -30624.244} C_VEL
LIN {X 0,Y 27.539,Z 475.383,A -85,B 0,C 180,E1 -30640.03,E2 -30640.03} C_VEL
LIN {X 0,Y 20.592,Z 476.543,A -85,B 0,C 180,E1 -30670.036,E2 -30670.036} C_VEL
LIN {X 0,Y 19.88,Z 476.698,A -85,B 0,C 180,E1 -30689.992,E2 -30689.992} C_VEL
LIN {X 0,Y 23.334,Z 476.081,A -85,B 0,C 180,E1 -30727.031,E2 -30727.031} C_VEL
LIN {X 0,Y 32.76,Z 474.321,A -85,B 0,C 180,E1 -30749.094,E2 -30749.094} C_VEL
LIN {X 0,Y 44.691,Z 471.397,A -85,B 0,C 180,E1 -30760.643,E2 -30760.643} C_VEL
LIN {X 0,Y 57.63,Z 467.238,A -85,B 0,C 180,E1 -30767.301,E2 -30767.301} C_VEL
LIN {X 0,Y 71.054,Z 461.735,A -85,B 0,C 180,E1 -30771.517,E2 -30771.517} C_VEL
LIN {X 0,Y 84.751,Z 454.739,A -85,B 0,C 180,E1 -30774.299,E2 -30774.299} C_VEL
LIN {X 0,Y 92.479,Z 450.074,A -85,B 0,C 180,E1 -30775.642,E2 -30775.642} C_VEL
LIN {X 0,Y 94.435,Z 448.738,A -85,B 0,C 180,E1 -30776.801,E2 -30776.801} C_VEL
LIN {X 0,Y 95.004,Z 448.231,A -85,B 0,C 180,E1 -30780,E2 -30780} C_VEL
LIN {X 0,Y 94.235,Z 448.816,A -85,B 0,C 180,E1 -30784.278,E2 -30784.278} C_VEL
LIN {X 0,Y 91.741,Z 450.461,A -85,B 0,C 180,E1 -30785.223,E2 -30785.223} C_VEL
LIN {X 0,Y 77.988,Z 458.239,A -85,B 0,C 180,E1 -30787.593,E2 -30787.593} C_VEL
LIN {X 0,Y 64.462,Z 464.426,A -85,B 0,C 180,E1 -30791.137,E2 -30791.137} C_VEL
LIN {X 0,Y 51.258,Z 469.201,A -85,B 0,C 180,E1 -30796.321,E2 -30796.321} C_VEL
LIN {X 0,Y 38.775,Z 472.692,A -85,B 0,C 180,E1 -30805.02,E2 -30805.02} C_VEL
LIN {X 0,Y 27.828,Z 474.993,A -85,B 0,C 180,E1 -30820.752,E2 -30820.752} C_VEL
LIN {X 0,Y 20.77,Z 476.157,A -85,B 0,C 180,E1 -30850.23,E2 -30850.23} C_VEL
LIN {X 0,Y 19.973,Z 476.31,A -85,B 0,C 180,E1 -30870.008,E2 -30870.008} C_VEL
LIN {X 0,Y 23.562,Z 475.741,A -85,B 0,C 180,E1 -30906.632,E2 -30906.632} C_VEL
LIN {X 0,Y 32.963,Z 474.047,A -85,B 0,C 180,E1 -30928.53,E2 -30928.53} C_VEL
LIN {X 0,Y 44.892,Z 471.187,A -85,B 0,C 180,E1 -30939.945,E2 -30939.945} C_VEL
LIN {X 0,Y 57.795,Z 467.095,A -85,B 0,C 180,E1 -30946.618,E2 -30946.618} C_VEL
LIN {X 0,Y 71.18,Z 461.671,A -85,B 0,C 180,E1 -30950.887,E2 -30950.887} C_VEL
LIN {X 0,Y 84.845,Z 454.758,A -85,B 0,C 180,E1 -30953.732,E2 -30953.732} C_VEL
LIN {X 0,Y 91.728,Z 450.678,A -85,B 0,C 180,E1 -30954.9,E2 -30954.9} C_VEL
LIN {X 0,Y 94.21,Z 449.048,A -85,B 0,C 180,E1 -30955.721,E2 -30955.721} C_VEL
LIN {X 0,Y 94.556,Z 448.737,A -85,B 0,C 180,E1 -30957.853,E2 -30957.853} C_VEL
LIN {X 0,Y 94.139,Z 448.99,A -85,B 0,C 180,E1 -30958.952,E2 -30958.952} C_VEL
LIN {X 0,Y 92.566,Z 449.993,A -85,B 0,C 180,E1 -30960.039,E2 -30960.039} C_VEL
LIN {X 0,Y 89.508,Z 451.903,A -85,B 0,C 180,E1 -30960.968,E2 -30960.968} C_VEL
LIN {X 0,Y 82.642,Z 455.809,A -85,B 0,C 180,E1 -30961.433,E2 -30961.433} C_VEL
LIN {X 0,Y 76.744,Z 458.818,A -85,B 0,C 180,E1 -30961.818,E2 -30961.818} C_VEL
LIN {X 0,Y 63.407,Z 464.718,A -85,B 0,C 180,E1 -30963.989,E2 -30963.989} C_VEL
LIN {X 0,Y 49.628,Z 469.501,A -85,B 0,C 180,E1 -30967.548,E2 -30967.548} C_VEL
LIN {X 0,Y 36.192,Z 473.007,A -85,B 0,C 180,E1 -30973.833,E2 -30973.833} C_VEL
LIN {X 0,Y 23.581,Z 475.313,A -85,B 0,C 180,E1 -30986.594,E2 -30986.594} C_VEL
LIN {X 0,Y 14.096,Z 476.474,A -85,B 0,C 180,E1 -31020.082,E2 -31020.082} C_VEL
LIN {X 0,Y 12.767,Z 476.628,A -85,B 0,C 180,E1 -31049.988,E2 -31049.988} C_VEL
LIN {X 0,Y 18.139,Z 476.012,A -85,B 0,C 180,E1 -31100.78,E2 -31100.78} C_VEL
LIN {X 0,Y 29.723,Z 474.251,A -85,B 0,C 180,E1 -31121.031,E2 -31121.031} C_VEL
LIN {X 0,Y 42.851,Z 471.326,A -85,B 0,C 180,E1 -31129.731,E2 -31129.731} C_VEL
LIN {X 0,Y 56.488,Z 467.168,A -85,B 0,C 180,E1 -31134.417,E2 -31134.417} C_VEL
LIN {X 0,Y 70.355,Z 461.664,A -85,B 0,C 180,E1 -31137.294,E2 -31137.294} C_VEL
LIN {X 0,Y 84.341,Z 454.668,A -85,B 0,C 180,E1 -31139.177,E2 -31139.177} C_VEL
LIN {X 0,Y 87.603,Z 452.788,A -85,B 0,C 180,E1 -31139.549,E2 -31139.549} C_VEL
LIN {X 0,Y 88.903,Z 452.034,A -85,B 0,C 180,E1 -31140.001,E2 -31140.001} C_VEL
LIN {X 0,Y 87.618,Z 452.764,A -85,B 0,C 180,E1 -31141.164,E2 -31141.164} C_VEL
LIN {X 0,Y 73.884,Z 459.981,A -85,B 0,C 180,E1 -31142.882,E2 -31142.882} C_VEL
LIN {X 0,Y 60.016,Z 465.815,A -85,B 0,C 180,E1 -31145.55,E2 -31145.55} C_VEL
LIN {X 0,Y 49.718,Z 469.272,A -85,B 0,C 180,E1 -31148.339,E2 -31148.339} C_VEL
LIN {X 0,Y 36.336,Z 472.762,A -85,B 0,C 180,E1 -31154.76,E2 -31154.76} C_VEL
LIN {X 0,Y 23.79,Z 475.063,A -85,B 0,C 180,E1 -31167.608,E2 -31167.608} C_VEL
LIN {X 0,Y 14.273,Z 476.226,A -85,B 0,C 180,E1 -31200.514,E2 -31200.514} C_VEL
LIN {X 0,Y 12.87,Z 476.379,A -85,B 0,C 180,E1 -31230.012,E2 -31230.012} C_VEL
LIN {X 0,Y 18.341,Z 475.81,A -85,B 0,C 180,E1 -31280.04,E2 -31280.04} C_VEL
LIN {X 0,Y 29.862,Z 474.116,A -85,B 0,C 180,E1 -31300.299,E2 -31300.299} C_VEL
LIN {X 0,Y 42.967,Z 471.256,A -85,B 0,C 180,E1 -31308.946,E2 -31308.946} C_VEL
LIN {X 0,Y 56.57,Z 467.164,A -85,B 0,C 180,E1 -31313.673,E2 -31313.673} C_VEL
LIN {X 0,Y 70.402,Z 461.739,A -85,B 0,C 180,E1 -31316.642,E2 -31316.642} C_VEL
LIN {X 0,Y 84.364,Z 454.826,A -85,B 0,C 180,E1 -31318.563,E2 -31318.563} C_VEL
LIN {X 0,Y 87.643,Z 452.944,A -85,B 0,C 180,E1 -31318.918,E2 -31318.918} C_VEL
LIN {X 0,Y 88.923,Z 452.217,A -85,B 0,C 180,E1 -31319.999,E2 -31319.999} C_VEL
LIN {X 0,Y 87.629,Z 452.966,A -85,B 0,C 180,E1 -31320.382,E2 -31320.382} C_VEL
LIN {X 0,Y 76.744,Z 458.818,A -85,B 0,C 180,E1 -31321.818,E2 -31321.818} C_VEL
LIN {X 0,Y 69.185,Z 462.323,A -85,B 0,C 180,E1 -31322.372,E2 -31322.372} C_VEL
LIN {X 0,Y 56.208,Z 467.261,A -85,B 0,C 180,E1 -31321.947,E2 -31321.947} C_VEL
LIN {X 0,Y 45.59,Z 470.534,A -85,B 0,C 180,E1 -31321.348,E2 -31321.348} C_VEL
LIN {X 0,Y 37.517,Z 472.472,A -85,B 0,C 180,E1 -31321.874,E2 -31321.874} C_VEL
LIN {X 0,Y 34.829,Z 473.002,A -85,B 0,C 180,E1 -31322.526,E2 -31322.526} C_VEL
LIN {X 0,Y 21.359,Z 475.244,A -85,B 0,C 180,E1 -31329.157,E2 -31329.157} C_VEL
LIN {X 0,Y 8.679,Z 476.405,A -85,B 0,C 180,E1 -31355.897,E2 -31355.897} C_VEL
LIN {X 0,Y 5.665,Z 476.559,A -85,B 0,C 180,E1 -31409.973,E2 -31409.973} C_VEL
LIN {X 0,Y 14.703,Z 475.942,A -85,B 0,C 180,E1 -31482.904,E2 -31482.904} C_VEL
LIN {X 0,Y 28.22,Z 474.181,A -85,B 0,C 180,E1 -31494.913,E2 -31494.913} C_VEL
LIN {X 0,Y 42.167,Z 471.256,A -85,B 0,C 180,E1 -31499.385,E2 -31499.385} C_VEL
LIN {X 0,Y 45.088,Z 470.509,A -85,B 0,C 180,E1 -31500.001,E2 -31500.001} C_VEL
LIN {X 0,Y 42.179,Z 471.24,A -85,B 0,C 180,E1 -31501.523,E2 -31501.523} C_VEL
LIN {X 0,Y 28.265,Z 474.128,A -85,B 0,C 180,E1 -31506.034,E2 -31506.034} C_VEL
LIN {X 0,Y 14.811,Z 475.854,A -85,B 0,C 180,E1 -31518.41,E2 -31518.41} C_VEL
LIN {X 0,Y 5.759,Z 476.448,A -85,B 0,C 180,E1 -31590.027,E2 -31590.027} C_VEL
LIN {X 0,Y 14.811,Z 475.879,A -85,B 0,C 180,E1 -31661.661,E2 -31661.661} C_VEL
LIN {X 0,Y 28.267,Z 474.185,A -85,B 0,C 180,E1 -31674.045,E2 -31674.045} C_VEL
LIN {X 0,Y 42.184,Z 471.325,A -85,B 0,C 180,E1 -31678.524,E2 -31678.524} C_VEL
LIN {X 0,Y 45.056,Z 470.601,A -85,B 0,C 180,E1 -31679.999,E2 -31679.999} C_VEL
LIN {X 0,Y 34.829,Z 473.002,A -85,B 0,C 180,E1 -31682.526,E2 -31682.526} C_VEL
LIN {X 0,Y 33.219,Z 474.97,A -85,B 0,C 180,E1 -31683.049,E2 -31683.049} C_VEL
LIN {X 0,Y 33.219,Z 600,A -85,B 0,C 180,E1 -31683.049,E2 -31683.049} C_VEL
LIN {X 0,Y 33.219,Z 600,A -85,B 0,C 180,E1 -31683.049,E2 -31683.049}

QRS_NEXT_CUT()

QRS_NEXT()
QRS_HOME()

END
